RoboDK station: robot_vesion.rdk

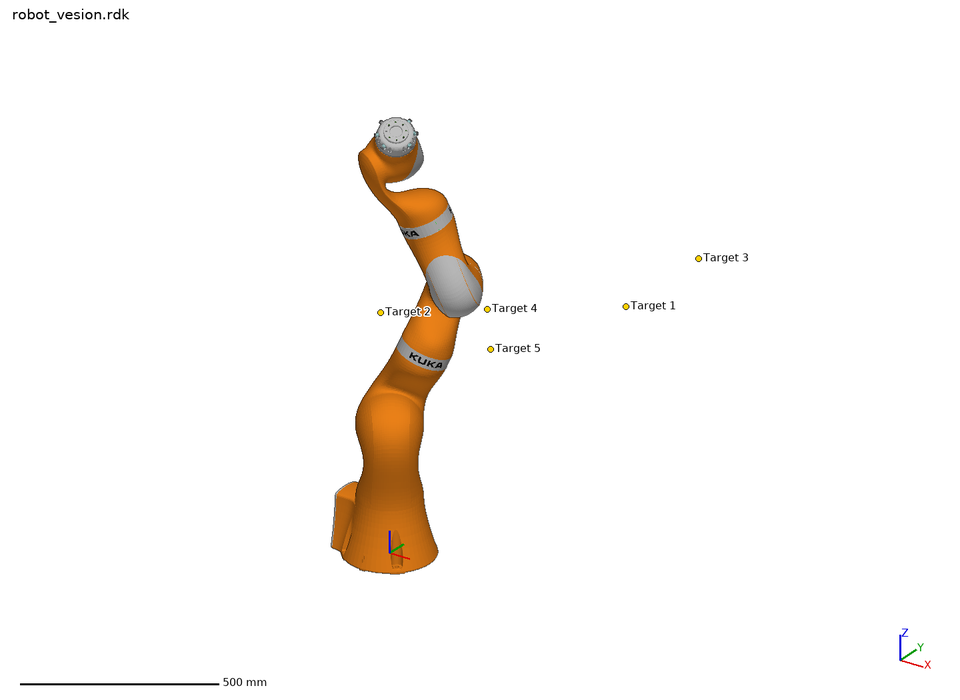
[picture v0: the station drawn from its stored meshes, robots at their saved joint values, targets as dots, program paths as lines]
Station kuka (saved by RoboDK 5.6.0). Poses are relative to the parent item; angles as X-Y-Z fixed-axis rotations.
  - frame KUKA LBR iiwa 14 R820 Base at (0, 0, 0) mm
    - robot KUKA LBR iiwa 14 R820: 7 axes, payload 14 kg, reach 1180 mm, repeatability 0.15 mm, weight 29.9 kg
        modified DH rows (alpha deg, a mm, theta deg, d mm): 0, 0, 0, 360; -90, 0, 0, 0; 90, 0, 0, 420; -90, 0, 0, 0; 90, 0, 0, 400; -90, 0, 0, 0; 90, 0, 0, 90
        joint limits [-170, -120, -170, -120, -170, -120, -175] to [170, 120, 170, 120, 170, 120, 175]; home [0, 0, 0, -90, 0, 0, 0]; saved at [37.916, 23.308, 0, -45.549, -65.153, 42.625, 57.817]
      - tool Tool 1, TCP at (0, 0, 200) mm
    - target Target 1 (Cartesian target) at (725, 0, 890) mm, rotated rx 0 ry 90 rz 0 deg; joints [0, -90, 90, 0, 0, 0] of KUKA LBR iiwa 14 R820
    - target Target 2 (Cartesian target) at (240.17, -379.9, 890) mm, rotated rx 0 ry 90 rz 0 deg; joints [95.985, -97.913, 97.321, -90.062, 95.985, 89.406] of KUKA LBR iiwa 14 R820
    - target Target 3 (Cartesian target) at (715.43, 331.38, 890) mm, rotated rx 0 ry 90 rz 0 deg; joints [-37.273, -76.872, 75.248, -92.133, -37.303, 92.681] of KUKA LBR iiwa 14 R820
    - target Target 4 (Cartesian target) at (318.63, -25.44, 780) mm, rotated rx 0 ry 90 rz 0 deg; joints [-41.627, -51.534, 0, -118.153, -114.063, -46.678, 123.058] of KUKA LBR iiwa 14 R820
    - target Target 5 (Cartesian target) at (456.36, -209.07, 780) mm, rotated rx 0 ry 90 rz 0 deg; joints [-51.49, -18.354, 0, -105.292, -92.434, -51.555, 93.911] of KUKA LBR iiwa 14 R820
  - Python program Prog1 (listed below)
  - Python program Prog2 (listed below)
  - Python program Prog3 (listed below)

--- Python program Prog1 ---
# Type help("robodk.robolink") or help("robodk.robomath") for more information
# Press F5 to run the script
# Documentation: https://robodk.com/doc/en/RoboDK-API.html
# Reference:     https://robodk.com/doc/en/PythonAPI/robodk.html
# Note: It is not required to keep a copy of this file, your Python script is saved with your RDK project
# Draw a hexagon around Target 1
from robolink import *    # RoboDK's API
from robodk.robolink import *
      # Math toolbox for robots

# Start the RoboDK API:
RDK = Robolink()

# Get the robot (first robot found):
robot = RDK.Item('', ITEM_TYPE_ROBOT)

# Get the reference target by name:
target = RDK.Item('Target 1')
target2 = RDK.Item('Target 2')
target3 = RDK.Item('Target 3')
target_pose = target.Pose()
xyz_ref = target_pose.Pos()

# Move the robot to the reference point:
robot.MoveJ(target)
robot.MoveJ(target2)
robot.MoveJ(target3)

## Control por Visión ##
# El programa mueve el robot de uno de los targets definidos al otro en funcion de los dedos que se levanten(índice/índice+corazón)
import cv2 as cv
import mediapipe as mp
import time
import math


def findPos(img,results,handNumb=0,draw=False,palmLM = False, drawPalm = False):

    lmList = []
    if results.multi_hand_landmarks:
        myHand = results.multi_hand_landmarks[handNumb]
        for i,lm in enumerate(myHand.landmark):
            h,w,c=img.shape
            cx,cy,cz=int(lm.x*w),int(lm.y*h),lm.z
            lmList.append([i,cx,cy,cz])
            if draw:
                cv.circle(img, (cx,cy), 5, (255,255,0), cv.FILLED)
        if palmLM:
            palmMarks = [0, 1, 5, 9, 13, 17]
            palmX, palmY, palmZ = 0, 0, 0
            for id in palmMarks:
                palmX += lmList[id][1]
                palmY += lmList[id][2]
                palmZ += lmList[id][3]
            palm = [21, int(palmX/6), int(palmY/6), palmZ/6]
            lmList.append(palm)
            if drawPalm:
                cv.circle(img, (palm[1],palm[2]), 5, (255,255,0), cv.FILLED)
    return lmList

def lmDistance(lm1,lm2):
    dx = lm2[1]-lm1[1]
    dy = lm2[2]-lm1[2]
    dist = math.sqrt((dx**2)+(dy**2))
    return int(dist)

def fingersState(lmList):
    fingersUp = []
    fingersCount = 0
    tipIds = [4, 8, 12, 16, 20]
    for id in tipIds:
        if id == 4:
            distP = lmDistance(lmList[id],lmList[17])
            distF = lmDistance(lmList[id-2],lmList[17])
        else:
            distP = lmDistance(lmList[id],lmList[0])
            distF = lmDistance(lmList[id-2],lmList[0])
        if distP > distF:
            fingersCount += 1
            fingersUp.append(1)
        else:
            fingersUp.append(0)
    return fingersUp, fingersCount


cap = cv.VideoCapture(0)
mpHands = mp.solutions.hands
hands = mpHands.Hands()
mpDraw = mp.solutions.drawing_utils

pTime = 0
cTime = 0


while True:
    success , frame = cap.read()
    frame = cv.flip(frame,1)
    frameRGB=cv.cvtColor(frame,cv.COLOR_BGR2RGB)
    results=hands.process(frameRGB)
    lmList = findPos(frame,results,handNumb=0,draw=True,palmLM = False, drawPalm = False)
    if len(lmList) != 0:
        fingerState, fingersCount = fingersState(lmList)
        cv.putText(frame,'fingerState:'+str(fingerState),(20,100),cv.FONT_HERSHEY_COMPLEX,
                   0.5,(0,255,0),thickness=1)
        if fingerState == [0,1,0,0,0]:
            cv.putText(frame,'Target 1',(200,300),cv.FONT_HERSHEY_COMPLEX,
                   1,(0,0,255),thickness=1)
            robot.MoveJ(target)
            robot.RunInstruction('Program_Done')
        if fingerState == [0,1,1,0,0]:
            cv.putText(frame,'Target 2',(200,300),cv.FONT_HERSHEY_COMPLEX,
                   1,(0,0,255),thickness=1)
            robot.MoveJ(target2)
            robot.RunInstruction('Program_Done')
        if fingerState == [0,1,1,1,0]:
            cv.putText(frame,'Target 3 ',(200,300),cv.FONT_HERSHEY_COMPLEX,
                   1,(0,0,255),thickness=1)
            robot.MoveJ(target3)
            robot.RunInstruction('Program_Done')



    cTime = time.time()
    fps = 1/(cTime-pTime)
    pTime = cTime

    cv.putText(frame,'fps:'+str(int(fps)),(20,40),cv.FONT_HERSHEY_COMPLEX,
    1,(0,255,0),thickness=2)

    cv.imshow('Video',frame)
    if cv.waitKey(20) & 0xFF==27:
        break


cap.release()
cv.destroyAllWindows()

# Trigger a program call at the end of the movement
robot.RunInstruction('Program_Done')

--- Python program Prog2 ---
import cv2
from robodk.robolink import *
from robodk import *

# Initialize RoboDK
RDK = Robolink()

# Load the KUKA robot
robot = RDK.Item('KUKA Robot')

# Define target positions [x, y, z] (modify these)
target_positions = [
    [1000, 200, 300],
    [800, 400, 500],
    [600, 600, 700]
]

# Initialize camera (OpenCV)
camera = cv2.VideoCapture(0)  # Use the appropriate camera index

while True:
    # Capture a frame from the camera
    ret, frame = camera.read()

    # ... Finger detection code (same as before)

    # Move the robot to the detected number of fingers (targets)
    if finger_count >= 1 and finger_count <= 3:
        target_index = finger_count - 1
        target_pose = Pose(target_positions[target_index])
        robot.MoveJ(target_pose)

    cv2.imshow('Camera Feed', frame)

    # Exit the loop if the 'q' key is pressed
    if cv2.waitKey(1) & 0xFF == ord('q'):
        break

# Release the camera and close windows
camera.release()
cv2.destroyAllWindows()

--- Python program Prog3 ---
import math
import cv2
import numpy as np
import mediapipe as mp
from robodk.robolink import *

RDK = Robolink()
import time

frameWidth = 640
frameHeight = 480

cpx=int(frameWidth/2)
cpy=int(frameHeight/2)

maxlen=120
minlen=30

open=85
close=0

robot=RDK.Item('',ITEM_TYPE_ROBOT)


target = RDK.Item('Target 1')
target2 = RDK.Item('Target 2')
target3 = RDK.Item('Target 3')
target4 = RDK.Item('Target 4')
target5 = RDK.Item('Target 5')
target_pose = target.Pose()
xyz_ref = target_pose.Pos()



tips = [4,8,12,16,20]
cap=cv2.VideoCapture(0)
cap.set(3,frameWidth)
cap.set(4,frameHeight)

mphands=mp.solutions.hands

hands=mphands.Hands()

mpdraw=mp.solutions.drawing_utils

#draw=mp.solutions.drawing_utils
draw=mp.solutions.drawing_styles
ptime=0
ctime=0

def finger_fun(limx,limy,tips):
    finger_state=[]

    for id in tips :
        if id ==4:
            if limx[17]-limx[4] > 100:
                finger_state.append(1)

            else:finger_state.append(0)
        else:
            if limy[id] < limy[id-2] :
             finger_state.append(1)
            else:finger_state.append(0)

    return finger_state

while True :

    _ ,img =cap.read()
    img = cv2.flip(img,1)
    cv2.circle(img,(cpx, cpy),15,(255,0,0),cv2.FILLED)

    imgrgb=cv2.cvtColor(img,cv2.COLOR_BGR2RGB)
    results=hands.process(imgrgb)

    if results.multi_hand_landmarks :
        for handlms in results.multi_hand_landmarks :
            lim_list=[]
            limx=[]
            limy=[]
            for id ,lm in enumerate(handlms.landmark):
                lim_list.append(lm)
                h,w,c= img.shape
                cx=int(w * lm.x)
                cy=int(h * lm.y)
                #print(cx,cy)
                limx.append(cx)
                limy.append(cy)

                mpdraw.draw_landmarks(img, handlms,mphands.HAND_CONNECTIONS)




        finger=finger_fun(limx,limy,tips)
        print(finger)


        if finger == [0,1,0,0,0]:
            cv2.putText(img,'Target 1',(200,300),cv2.FONT_HERSHEY_COMPLEX,
                   1,(0,0,255),thickness=1)
            robot.MoveJ(target)
            robot.RunInstruction('Program_Done')
        if finger == [0,1,1,0,0]:
            cv2.putText(img,'Target 2',(200,300),cv2.FONT_HERSHEY_COMPLEX,
                   1,(0,0,255),thickness=1)
            robot.MoveJ(target2)
            robot.RunInstruction('Program_Done')
        if finger == [0,1,1,1,0]:
            cv2.putText(img,'Target 3 ',(200,300),cv2.FONT_HERSHEY_COMPLEX,
                   1,(0,0,255),thickness=1)
            robot.MoveJ(target3)
            robot.RunInstruction('Program_Done')


        if finger == [0,1,1,1,1]:
            cv2.putText(img,'Target 4 ',(200,300),cv2.FONT_HERSHEY_COMPLEX,
                   1,(0,0,255),thickness=1)
            robot.MoveJ(target4)
            robot.RunInstruction('Program_Done')

        if finger == [1,1,1,1,1]:
            cv2.putText(img,'Target 5 ',(200,300),cv2.FONT_HERSHEY_COMPLEX,
                   1,(0,0,255),thickness=1)
            robot.MoveJ(target5)
            robot.RunInstruction('Program_Done')









    ctime=time.time()
    fps=1/(ctime-ptime)
    ptime=ctime
    #print(fps)

    cv2.putText(img,str(int(fps)),(50,450),cv2.FONT_HERSHEY_PLAIN,3,(255,0,0),3)
    cv2.imshow('first',img)
    cv2.waitKey(1)
